PROGRAM FBD
VAR
	count : INT := 0;
	reset : BOOL := FALSE;
END_VAR

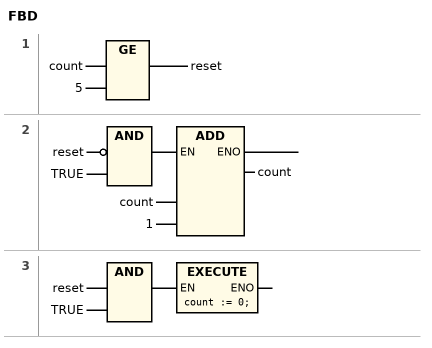
// NETWORK 1
reset := count >= 5;

// NETWORK 2
IF NOT reset AND TRUE THEN count := count + 1; END_IF

// NETWORK 3
IF reset AND TRUE THEN count := 0; END_IF

END_PROGRAM

(* stored: Version 1.1.0.1, ProductVersion 3.1.4024.12
   POU FBD: Id {e81c59f2-b698-4ecb-8daf-30291b7b4191}, SpecialFunc None *)
